// Hardware-linked primitives for FB_DigitalInput. Link at instance site via
// {attribute 'TcLinkTo' := '.io.inSignal := TIID^...'}.
TYPE ST_DigitalInput_IO :
STRUCT
    inSignal AT %I* : BOOL;
END_STRUCT
END_TYPE

(* stored: Version 1.1.0.1, ProductVersion 3.1.4026.12
   DUT ST_DigitalInput_IO: Id {b0100001-0003-0000-0000-000000000001} *)
